PROGRAM PRG_Compilation
VAR
	fbLoggerElement				: FB_BaseLoggerElement;
	fbLoggerElementDecorator	: FB_BaseLoggerElementDecoratorParent (fbToDecorate := fbLoggerElement);
	fbComponent					: FB_BaseComponent;
	fbComponentDecorator		: FB_BaseComponentDecoratorParent (fbToDecorate := fbComponent);
	fbControlElement			: FB_BaseControlElement;
	fbControlElementDecorator	: FB_BaseControlElementDecoratorParent (fbToDecorate := fbControlElement);
	fbGroupElement				: FB_BaseGroupElement;
	fbGroupElementDecorator		: FB_BaseGroupElementDecoratorParent (fbToDecorate := fbGroupElement);
	fbTopElement				: FB_BaseTopElement;
	fbTopElementDecorate		: FB_BaseTopElementDecoratorParent (fbToDecorate := fbTopElement);
END_VAR

END_PROGRAM

(* stored: Version 1.1.0.1
   POU PRG_Compilation: Id {824d9806-ef98-4594-8f89-7dfa640c0d27}, SpecialFunc None *)
